// TwinCAT 3 PLC project
// libraries:
//   SyntheticLibrary
// project tree:
//   GVLs/ Plant.TcGVL
//   POUs/ MAIN.TcPOU

// ---- GVLs/Plant.TcGVL
VAR_GLOBAL
  PumpAlpha : FB_Device;
  FlowValue : REAL;
  ValveCommand : BOOL := FALSE;
END_VAR

// ---- POUs/MAIN.TcPOU
PROGRAM MAIN
VAR
  LocalPermit : BOOL;
END_VAR


Plant.PumpAlpha(Start := LocalPermit);
Plant.ValveCommand := LocalPermit;
// Plant.DeprecatedValve := TRUE;

END_PROGRAM
